// TIA Portal V19 export
TYPE "typeSafetyDrive"
// Safety status of drive
// stored: Access Published, IsFailsafeCompliant true, Namespace Safety
   STRUCT
      safetyFault { ExternalWritable := 'False'} : Bool;   // Safety fault in the drive 0: Fault-free operation
      stoActive { ExternalWritable := 'False'} : Bool;   // If false STO triggered
      ss1Active { ExternalWritable := 'False'} : Bool;   // If false SS1 triggered
      slsActive { ExternalWritable := 'False'} : Bool;   // If false SLS triggered
   END_STRUCT;
END_TYPE
